{attribute 'qualified_only'}
{attribute 'strict'}
TYPE Direction :
(
    Position := MC_Positive_Direction,
    ShortestWay := MC_Shortest_Way ,
    Negative := MC_Negative_Direction,
    Current := MC_Current_Direction,
	Undefined := MC_Undefined_Direction
) INT;
END_TYPE

(* stored: Version 1.1.0.1, ProductVersion 3.1.4024.12
   DUT Direction: Id {b86ed26b-71b9-09e1-223a-02e4f5a72de9} *)
